Yaskawa INFORM job: GO-TO-STATION-2-FRONT.JBI

/JOB
//NAME GO-TO-STATION-2-FRONT
//POS
///NPOS 2,0,0,1,0,0
///TOOL 0
///POSTYPE PULSE
///PULSE
C00000=123306,-222014,-26224,0,-132993,0
C00001=115325,-31618,-8148,-84937,-113078,91751
P00000=0,-222014,-26224,0,-132993,0
//INST
///DATE 2018/09/17 10:40
///ATTR SC,RW
///GROUP1 RB1
NOP
MOVJ P0000 VJ=50.00
'*****
SETREG MREG#(1) 1
MOVJ C00000 VJ=25.00
'*****
SETREG MREG#(1) 100
MOVJ C00001 VJ=25.00
'*****
SETREG MREG#(1) 111
END
